INTERFACE I_CyclicFB EXTENDS I_BaseFB

METHOD CyclicLogic
VAR_INPUT
END_VAR
END_METHOD

PROPERTY InitComplete : BOOL
GET
END_GET
END_PROPERTY

END_INTERFACE

(* stored: Version 1.1.0.1, ProductVersion 3.1.4024.12
   Itf I_CyclicFB: Id {c343820d-f6ec-4190-bd94-c0df0564e74d}
   Method CyclicLogic: Id {179830e2-1348-4010-bbbb-e80846a4b45c}
   Property InitComplete: Id {0969f1a6-d235-40bf-acf5-1bc6beb1f959}
   Get Get: Id {acee56f7-5098-492f-a278-c45223dafddc} *)
